Fanuc KAREL source: ka00134.KL

-- PROVISIONAL review KL for V940-1; original PC SHA256 ffc31fead4807119cd0f7a2b3ba26f74cbd5fced47d55f2f1d2796b68e2b6b49
-- Incomplete behavior may be omitted. Consult companion uncertainty JSON. Do not deploy.
PROGRAM KA00134
%NOLOCKGROUP
VAR
  DST : REAL
-- UNRESOLVED_DECL SRC type=002017
BEGIN
  -- V9_ZERO_TABLE_METADATA_HINT layout=0001; no indexed target words; source/name/runtime held
  -- UNRESOLVED_PC offsets 5-19; opcodes 2E,22,9D,33,B4
  -- UNRESOLVED_PC offsets 24-40; opcodes 22,9D,33,B3,64,23
  -- UNRESOLVED_PC offsets 45-49; opcodes 7F
END KA00134
